INTERFACE I_State

PROPERTY CurrentState : STRING
GET
END_GET
END_PROPERTY

METHOD ErrorGone
VAR_INPUT
END_VAR
END_METHOD

METHOD ErrorOccured
VAR_INPUT
END_VAR
END_METHOD

METHOD StartProcess
VAR_INPUT
END_VAR
END_METHOD

METHOD StopProcess
VAR_INPUT
END_VAR
END_METHOD

END_INTERFACE

(* stored: Version 1.1.0.1
   Itf I_State: Id {7e4bdf46-6fe1-4ad5-a34a-a1394a911493}
   Property CurrentState: Id {e320703d-028e-4b7d-8ba4-9c96866fa8f7}
   Get Get: Id {37560c9c-f8ec-4fee-adbd-a23a55a1b79c}
   Method ErrorGone: Id {196b2164-7aa9-45e3-9956-d81f1df78f2f}
   Method ErrorOccured: Id {7a0f543e-620b-466b-bef1-3ef60125ce50}
   Method StartProcess: Id {005f5047-dcca-496b-8621-253e9d3ed68d}
   Method StopProcess: Id {02d47221-6d9c-486f-a29d-a0de3e13ac93} *)
